// TIA Portal V19 export
TYPE "LAF_typeSequenceStep"
// Step
// stored: Access Published
   STRUCT
      "step" { ExternalWritable := 'False'} : DInt;   // State number
      duration { ExternalWritable := 'False'} : LReal;   // Time stayed in that state
   END_STRUCT;
END_TYPE
